// TIA Portal V21 export
// export: Created 2000-01-01T00:00:00.0000000Z, ExportSetting None
TYPE "UDT_TankStatus"
TITLE = 液位控制系统数据结构
// 液位控制系统数据类型：罐体测量值、目标液位、上下限阈值、报警标志、运行计数。
// 通常实例化为全局 DB_TankStatus 供 FC_LevelControl / FC_Alarm 等读写。
   STRUCT
      Level { ExternalWritable := 'False'} : Real;   // 罐体当前液位（单位：%，0~100）
      TargetLevel : Real;   // 操作员设定的目标液位（HMI 可写）
      HighLimit : Real;   // 高液位报警阈值，默认 90%
      LowLimit : Real;   // 低液位报警阈值，默认 10%
      AlarmHigh { ExternalWritable := 'False'} : Bool;   // 高液位报警标志（FC_Alarm 锁存）
      AlarmLow { ExternalWritable := 'False'} : Bool;   // 低液位报警标志（FC_Alarm 锁存）
      CycleCount { ExternalWritable := 'False'} : DInt;   // 运行启动累计次数
   END_STRUCT;
END_TYPE
